FUNCTION_BLOCK EncodeINeredaAct (* Composite Function Block Type *)
  (* Standard: 61499-2 *)
  (* Version 0.0, 6/7/2026, Schneider Electric, template *)
  PACKAGE SE.Nereda;
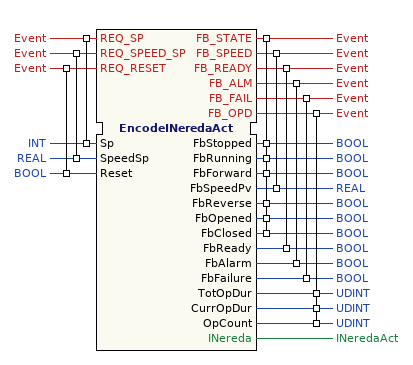
  EVENT_INPUT
    REQ_SP WITH Sp;
    REQ_SPEED_SP WITH SpeedSp;
    REQ_RESET WITH Reset;
  END_EVENT
  EVENT_OUTPUT
    FB_STATE WITH FbStopped, FbRunning, FbForward, FbReverse, FbOpened, FbClosed;
    FB_SPEED WITH FbSpeedPv;
    FB_READY WITH FbReady;
    FB_ALM WITH FbAlarm;
    FB_FAIL WITH FbFailure;
    FB_OPD WITH TotOpDur, CurrOpDur, OpCount;
  END_EVENT
  VAR_INPUT
    Sp : INT;
    SpeedSp : REAL;
    Reset : BOOL;
  END_VAR
  VAR_OUTPUT
    FbStopped : BOOL;
    FbRunning : BOOL;
    FbForward : BOOL;
    FbSpeedPv : REAL;
    FbReverse : BOOL;
    FbOpened : BOOL;
    FbClosed : BOOL;
    FbReady : BOOL;
    FbAlarm : BOOL;
    FbFailure : BOOL;
    TotOpDur : UDINT;
    CurrOpDur : UDINT;
    OpCount : UDINT;
  END_VAR
  PLUGS
    INereda : INeredaAct;
  END_PLUGS
  EVENT_CONNECTIONS
    INereda.9CD053F8408797ED TO FB_STATE;
    INereda.F846995A4121D865 TO FB_SPEED;
    INereda.CC753684FA882790 TO FB_READY;
    INereda.C79FD2A34D0395C5 TO FB_ALM;
    INereda.476AAA40EB7AA926 TO FB_FAIL;
    INereda.2DA8AEC15204E92D TO FB_OPD;
    REQ_SP TO INereda.0F1CDF9A9B4A227A;
    REQ_SPEED_SP TO INereda.1E00729184986247;
    REQ_RESET TO INereda.37BBC1F841739733;
  END_CONNECTIONS
  DATA_CONNECTIONS
    INereda.D83B5BDEFA4D797C TO FbStopped;
    INereda.B762734C094A7162 TO FbRunning;
    INereda.13E1B1B6EE0F07DB TO FbForward;
    INereda.3011FF733C667A56 TO FbReverse;
    INereda.790C5C3BA88E0AF5 TO FbSpeedPv;
    INereda.7F6CC7FEB9223DF3 TO FbOpened;
    INereda.A8D6C4A1FDCCA991 TO FbClosed;
    INereda.8A8A07EFCDA1443C TO FbReady;
    INereda.BDD69968F2D82EAF TO FbAlarm;
    INereda.6EEAF63EEE6021B6 TO FbFailure;
    INereda.C7F638DBF6B860D2 TO TotOpDur;
    INereda.9224E22E0E82A2D7 TO CurrOpDur;
    INereda.10624535249F94F3 TO OpCount;
    Sp TO INereda.710D7FC54EE3F35A;
    SpeedSp TO INereda.1BC103921BBFDA0B;
    Reset TO INereda.EA28053F07575F36;
  END_CONNECTIONS
END_FUNCTION_BLOCK
